DATA_BLOCK "DB_iPos_MC1"
{ S7_Optimized_Access := 'TRUE' }
VERSION : 0.1
NON_RETAIN
"FB_MachinePosition"

BEGIN

END_DATA_BLOCK

